        pointRx pPoint = {x=1198, y=151.559856, z=210.59, rx=87.981257, ry=172.229649, rz=-80.060298, fatherId=tTraj["test"].fFrame[0]}
        TrajectoryItem tSuper
          [0]
            string comment
            num distance
            InstrItem iInstr[3]
              [0]
                string sData
                string sType
              [1]
                string sData
                string sType
              [2]
                string sData
                string sType
            num moveType = 1
            num nMoveId
            num nStop
            num nTcpAction
            num nTime
            mdesc nom_speed = {accel=200, vel=450, decel=200, tmax=2000, blend=off}
            bool toStop = true
